TYPE TcaWorkpiecePlaceStatus : // EXTENDS ST_ComboboxEntry:
STRUCT
    ActionDescription : STRING(100);	
	Id : INT;
	Color: COLOR;
	PlaceStatus : eTcaWorkpiecePlaceStatus;
	Progress : eTcaWorkpiecePlaceProgress;
	
END_STRUCT
END_TYPE

(* stored: Version 1.1.0.1
   DUT TcaWorkpiecePlaceStatus: Id {7ca366c4-6112-4745-8034-11405d12e349} *)
